{attribute 'linkalways'} 
{attribute 'no_explicit_call' := 'This FB is a CLASS and must be accessed using methods or properties'}
{attribute 'enable_dynamic_creation'}
FUNCTION_BLOCK FINAL MAX_INT EXTENDS Node
VAR
	in1 : _INT(0);
	in2 : _INT(0);
	out : _INT(0);
END_VAR

METHOD PUBLIC Clone : I_Node
VAR
	pNode : POINTER TO MAX_INT;
END_VAR
pNode := __NEW(MAX_INT);
Clone := pNode^;
END_METHOD

METHOD FB_init : BOOL
VAR_INPUT
	bInitRetains : BOOL; // if TRUE, the retain variables are initialized (warm start / cold start)
	bInCopyCode : BOOL;  // if TRUE, the instance afterwards gets moved into the copy code (online change)
END_VAR
AddInput('in1',THIS^.in1);
AddInput('in2',THIS^.in2);
AddOutput('out', THIS^.out);
END_METHOD

METHOD PROTECTED OnExecute
VAR
END_VAR
out.Value := MAX(in1.Value, in2.Value);
END_METHOD

END_FUNCTION_BLOCK

(* stored: Version 1.1.0.1, ProductVersion 3.1.4024.15
   POU MAX_INT: Id {955ed7ab-731a-442b-89a6-9432dadd01d0}, SpecialFunc None
   Folder Constructor: Id {6bdfa6ce-0b14-4c22-b129-8e5ed69c171d}
   Method Clone: Id {9358db39-86b6-4b38-afbc-3df5b33c0f75}
   Method FB_init: Id {cff0fb10-a030-418d-bb14-8e3f1721b1bd}
   Method OnExecute: Id {207d30c9-b454-41b7-b560-eaace9636df7} *)
